METHOD PUBLIC IsFaulted : BOOL
VAR_INPUT
END_VAR
IsFaulted := (State = eGoodULNewStaState.eUnknown OR State = eGoodULNewStaState.eError);
END_METHOD

METHOD PUBLIC IsPalletHoldDownEngaged : BOOL
VAR_INPUT
END_VAR
IsPalletHoldDownEngaged := (GVL_IO.UL_3_XPalletHoldDownRetracted_Engaged AND NOT GVL_IO.UL_3_XPalletHoldDownExtended_Home);
IF (NOT IsPalletHoldDownEngaged) THEN
	Status.GoodUL_3_StatusMsg:= 'Good UL 3: Check Pallet Hold Down Sensors and then hit START';
END_IF
END_METHOD

METHOD PUBLIC IsPalletHoldDownFree : BOOL
VAR_INPUT
END_VAR
IsPalletHoldDownFree := (NOT GVL_IO.UL_3_XPalletHoldDownRetracted_Engaged AND GVL_IO.UL_3_XPalletHoldDownExtended_Home);
IF (NOT IsPalletHoldDownFree) THEN
	Status.GoodUL_3_StatusMsg := 'Good UL 3: Check Pallet Hold Down Sensors and then hit START';
END_IF
END_METHOD

PROPERTY PUBLIC Ready : BOOL
GET
IF (LotsData.Lot.GoodUnloadEnabled) THEN
	Ready := (State = eGoodULNewStaState.eReady);
ELSE
	Ready := (State = eGoodULNewStaState.eDisabledReady); 
END_IF
END_GET
END_PROPERTY

ACTION ResetDwellTimer:
DwellTimer(IN:=FALSE);
END_ACTION

METHOD PUBLIC ResetState : BOOL
VAR_INPUT
END_VAR
State := eGoodULNewStaState.eUnknown;
NextState := eGoodULNewStaState.eUnknown;
END_METHOD

PROPERTY PUBLIC Trigger : BOOL
SET
xTrigger := Trigger;
END_SET
END_PROPERTY

METHOD PUBLIC UpdateLotData : BOOL
VAR_INPUT
END_VAR
IF (PartsData.Status[VUT].Premium) THEN
	LotsData.Lot.CavityCounts[PartsData.Status[VUT].CavityNumber].PremiumCount := LotsData.Lot.CavityCounts[PartsData.Status[VUT].CavityNumber].PremiumCount +1;
ELSIF (PartsData.Status[VUT].Good) THEN
 	LotsData.Lot.CavityCounts[PartsData.Status[VUT].CavityNumber].GoodCount := LotsData.Lot.CavityCounts[PartsData.Status[VUT].CavityNumber].GoodCount + 1;
END_IF
LotsData.Lot.CavityCounts[PartsData.Status[VUT].CavityNumber].TotalCount := LotsData.Lot.CavityCounts[PartsData.Status[VUT].CavityNumber].TotalCount + 1;
 // reject parts shouldn't get here. If this station rejects something (e.g. faults out) then it barrel will go to reject station.
END_METHOD

METHOD PUBLIC UpdatePartData : BOOL
VAR_INPUT
END_VAR
PartsData.Status[VUT].UnloadTime := SYSTEMTIME_TO_STRING(Logging.fbCurrTime.systemTime);
PartsData.Status[VUT].OverallStatus := ePartStatus.eEmpty;
PartsData.Status[VUT].GoodUnload := TRUE;

// we will write data to CSV file over here 
IF (P_TextModeWrite.CurrWriteStep = 0) THEN 
	P_TextModeWrite.VehicleID := VUT;
	P_TextModeWrite.WriteData := TRUE;
END_IF
END_METHOD

PROPERTY PUBLIC VehicleUnderTest : BYTE
GET
VehicleUnderTest := VUT;
END_GET
SET
VUT := VehicleUnderTest;
END_SET
END_PROPERTY

END_FUNCTION_BLOCK

// ---- POUs/GoodULStation_4.TcPOU
FUNCTION_BLOCK PUBLIC GoodULStation_4
VAR_INPUT
END_VAR
VAR_OUTPUT
END_VAR
VAR
	xTrigger :BOOL := FALSE; // triggers processing
	State : eGoodULNewStaState := eGoodULNewStaState.eUnknown;
	NextState : eGoodULNewStaState := eGoodULNewStaState.eUnknown;
	ErrorReturnState : eGoodULNewStaState := eGoodULNewStaState.eUnknown;
	bFirst : BOOL := TRUE;
	VUT : BYTE; //VehicleID Under Station
	DwellTimer : TON;
	StateTimer : TON;
	GoodFullExcess: BYTE := 0;
END_VAR

IF (GVL_IO.MachineEStopped) THEN 
	State := eGoodULNewStaState.eUnknown;
	NextState := eGoodULNewStaState.eUnknown;
	Status.GoodUL_4_StatusMsg:= 'Good UL 4 Sta Unknown, Check AIR, E-STOP and Hit Start';
END_IF

CASE State OF
eGoodULNewStaState.eUnknown:
	Status.GoodUL_4_StatusMsg:= 'Good UL 4 Unknown, Check AIR, E-STOP and Hit Start';
    IF (GVL_IO.MC_XStartPB AND GVL_IO.MC_XAirPressureOK AND GVL_IO.MC_NotEStopped) THEN // wait for start button when powered up or PLC program restarted
		NextState := eGoodULNewStaState.eInit;	   
	END_IF
    

eGoodULNewStaState.eInit:
    Act_KnockPartOFF();
	Act_FreePalletHoldDown();
	ResetDwellTimer();
	NextState := eGoodULNewStaState.eHoming;
	

eGoodULNewStaState.eHoming:
	IF (IsPalletHoldDownFree()) THEN 
         NextState := eGoodULNewStaState.eReady;
	  END_IF
     DwellTimer(IN:=TRUE, PT:= T#10S);
     IF (DwellTimer.Q) THEN
		 ResetDwellTimer();
		 ErrorReturnState:= eGoodULNewStaState.eInit;
		 NextState := eGoodULNewStaState.eError;		 
	 END_IF	

eGoodULNewStaState.eReady:
	IF (xTrigger) THEN
		IF (NOT LotsData.Lot.AutoBaggerEnabled) THEN 
				Stations.fbRoutePlanner.P_GoodUnload_4_NextStaFlag := 5; 
				NextState := eGoodULNewStaState.eSendPalletHoldDownExtend;	
		ELSE
				NextState := eGoodULNewStaState.eCheckChuteCount;	
		END_IF	
		ResetDwellTimer();
	END_IF
	
	IF (NOT LotsData.Lot.GoodUnloadEnabled) THEN
		NextState :=  eGoodULNewStaState.eDisabledReady;	
	END_IF

eGoodULNewStaState.eDisabledReady:

	Act_KnockPartOFF();
	Act_FreePalletHoldDown();
	
    IF (LotsData.Lot.GoodUnloadEnabled) THEN 
		NextState := eGoodULNewStaState.eUnknown; // force the operator to hit the start button if station is enabled.
	END_IF
	
    IF (xTrigger) THEN // vehicles that have been previously commanded to come here before station was disabled 
		Stations.fbRoutePlanner.P_GoodUnload_4_NextStaFlag := 5; // send to reject after this process is complete
		NextState := eGoodULNewStaState.eDepart;
	END_IF
	
	Status.StationStauts[MM_CONST.GOOD_UL_4_STA_HMI_STATE] := OverallStationStatus.eDisabled;
	Status.GoodUL_4_StatusMsg:= 'Good UL1 Disabled and Clear for pallets to move';	

eGoodULNewStaState.eCheckChuteCount:
	IF  (Config.GoodCount2 < LotsData.Lot.QuantityInBag)  THEN
			Stations.fbRoutePlanner.P_GoodUnload_4_NextStaFlag := 5; // send to reject after this process is complete
			NextState := eGoodULNewStaState.eSendPalletHoldDownExtend;	          
 			GoodFullExcess:=0;  			
	ELSE  	
		    GoodFullExcess := GoodFullExcess +1;
			Stations.fbRoutePlanner.P_GoodUnload_4_NextStaFlag := 5; // send to reject after this process is complete
			NextState := eGoodULNewStaState.eDepart;
	END_IF 		
	IF (GoodFullExcess > 5) THEN 
		ErrorReturnState:= eGoodULNewStaState.eCheckChuteCount;		
		Status.GoodUL_4_StatusMsg:= 'No Drop Location for Part!Fix Bagger & Clear Chutes';
		NextState := eGoodULNewStaState.eError;		
    END_IF			


eGoodULNewStaState.eSendPalletHoldDownExtend:
	Act_EngagePalletHoldDown();
	ResetDwellTimer();
	NextState := eGoodULNewStaState.eCheckPalletHoldDownExtended;
	
eGoodULNewStaState.eCheckPalletHoldDownExtended:
   DwellTimer(IN:=TRUE, PT:= T#10S);	
   IF (IsPalletHoldDownEngaged()) THEN
        ResetDwellTimer();	   
		IF(GVL_IO.UL_4_XBarrelPresent (*OR TRUE*)) THEN /// enabled checking Part Present Sensor at Unload stations 051319 NAP
			NextState := eGoodULNewStaState.eKnockOffPart;
        ELSE
			NextState := eGoodULNewStaState.ePalletHoldDownRelease;	
		END_IF        
   END_IF      
   IF (DwellTimer.Q) THEN
		 ResetDwellTimer();
		 ErrorReturnState:= eGoodULNewStaState.eSendPalletHoldDownExtend;
		 NextState := eGoodULNewStaState.eError;		 
	END_IF
  
eGoodULNewStaState.eKnockoffPart:
	Act_KnockPartON();
	UpdateLotData();
	UpdatePartData();
	ResetDwellTimer();
	StateTimer(IN:=FALSE);	
	NextState := eGoodULNewStaState.eCheckPartKnockedOff;

eGoodULNewStaState.eCheckPartKnockedOff:
   StateTimer(IN:=TRUE, PT:= T#200MS);
   	IF (StateTimer.Q) THEN
   //IF (NOT(GVL_IO.UL_4_XBarrelPresent) ) THEN   
	   NextState := eGoodULNewStaState.ePalletHoldDownRelease;
	   Config.GoodCount2 := Config.GoodCount2 + 1;
	   DwellTimer(IN:=FALSE);
	   StateTimer(IN:=FALSE);
   END_IF
   DwellTimer(IN:= TRUE, PT:= T#10S);
   IF (DwellTimer.Q) THEN
	   ResetDwellTimer();
	   ErrorReturnState:= eGoodULNewStaState.eCheckPartKnockedOff;
	   Status.GoodUL_4_StatusMsg:= 'Good UL 4 Remove Part then Hit START';
   	   NextState := eGoodULNewStaState.eError;	
   END_IF   

eGoodULNewStaState.ePalletHoldDownRelease:
    Act_KnockPartOFF();
	Act_FreePalletHoldDown();
    ResetDwellTimer();	
	NextState := eGoodULNewStaState.ePalletHoldDownReleased;

eGoodULNewStaState.ePalletHoldDownReleased:	
	IF (IsPalletHoldDownFree()) THEN         
	    NextState := eGoodULNewStaState.eDepart;
    END_IF
	
   DwellTimer(IN:= TRUE, PT:= T#10S);
   IF (DwellTimer.Q) THEN
	   ResetDwellTimer();
	   ErrorReturnState:= eGoodULNewStaState.ePalletHoldDownRelease;	   
   	   NextState := eGoodULNewStaState.eError;	
   END_IF  
	
	
eGoodULNewStaState.eDepart:
    Stations.fbRoutePlanner.M_NotifyVehStaCmpl(StationIndex:= MM_CONST.GOOD_UL_4_STA, VehicleID := VUT);
	xTrigger := FALSE;
	IF (Stations.fbCycleControl.StopRequested) THEN
		NextState := eGoodULNewStaState.eStopActive;
	ELSE 
		NextState := eGoodULNewStaState.eReady;
    END_IF
	
eGoodULNewStaState.eStopActive:
	IF (NOT Stations.fbCycleControl.StopRequested) THEN
		NextState := eGoodULNewStaState.eInit;
    END_IF
	

eGoodULNewStaState.eError:
	IF (GVL_IO.MC_XStartPB) THEN
		NextState := ErrorReturnState;
		ErrorReturnState := eGoodULNewStaState.eUnknown;
	END_IF

END_CASE

IF (State <> NextState) THEN
	bFirst := TRUE;
	StateTimer(IN:=FALSE);
ELSE
	bFirst := FALSE;
END_IF

State := NextState;
AssignStationStatusForHMI();

ACTION Act_EngagePalletHoldDown:
GVL_IO.UL_4_YPalletHoldDownExtend_Home  := FALSE;
GVL_IO.UL_4_YPalletHoldDownRetract_Engage := TRUE;
END_ACTION

ACTION Act_FreePalletHoldDown:
GVL_IO.UL_4_YPalletHoldDownExtend_Home := TRUE;
GVL_IO.UL_4_YPalletHoldDownRetract_Engage := FALSE;
END_ACTION

ACTION Act_KnockPartOFF:
GVL_IO.UL_4_YRejectPushExtend := FALSE;
GVL_IO.UL_4_YRejectPushRetract := TRUE;
END_ACTION

ACTION Act_KnockPartON:
GVL_IO.UL_4_YRejectPushExtend := TRUE;
GVL_IO.UL_4_YRejectPushRetract := FALSE;
END_ACTION

METHOD PUBLIC AssignStationStatusForHMI : BOOL
VAR_INPUT
END_VAR
Status.StationsState[MM_CONST.GOOD_UL_4_STA_HMI_STATE] := State;
IF (NOT LotsData.Lot.GoodUnloadEnabled) THEN
	Status.StationStauts[MM_CONST.GOOD_UL_4_STA_HMI_STATE] := OverallStationStatus.eDisabled;
ELSE 
	CASE State OF 
	
	eGoodULNewStaState.eUnknown,eGoodULNewStaState.eError:
		Status.StationStauts[MM_CONST.GOOD_UL_4_STA_HMI_STATE] := OverallStationStatus.eError;
		
    eGoodULNewStaState.eInit,
	eGoodULNewStaState.eHoming:
	    Status.StationStauts[MM_CONST.GOOD_UL_4_STA_HMI_STATE] := OverallStationStatus.eHoming;
	
	eGoodULNewStaState.eReady,eGoodULNewStaState.eWaitForVehicleTrigger:
	     Status.StationStauts[MM_CONST.GOOD_UL_4_STA_HMI_STATE] := OverallStationStatus.eWaitingForParts;
		 
	eGoodULNewStaState.eDwell,
	eGoodULNewStaState.eSendPalletHoldDownExtend,
	eGoodULNewStaState.eCheckPalletHoldDownExtended,
	eGoodULNewStaState.ePalletReleaseExtend,
	eGoodULNewStaState.ePalletReleaseExtended,
	eGoodULNewStaState.eKnockoffPart,
	eGoodULNewStaState.eKnockoffExtended,
	eGoodULNewStaState.eCheckPartKnockedOff,
	eGoodULNewStaState.ePalletHoldDownRelease,
	eGoodULNewStaState.ePalletHoldDownReleased:
	    Status.StationStauts[MM_CONST.GOOD_UL_4_STA_HMI_STATE] := OverallStationStatus.eRunning;
	
	eGoodULNewStaState.eStopActive:
	    Status.StationStauts[MM_CONST.GOOD_UL_4_STA_HMI_STATE] := OverallStationStatus.eCycleStop;
    	
	
    ELSE;	
	END_CASE
END_IF
END_METHOD

METHOD PUBLIC ClearVehicleTrigger : BOOL
VAR_INPUT
END_VAR
xTrigger := FALSE;
END_METHOD

METHOD PUBLIC IsFaulted : BOOL
VAR_INPUT
END_VAR
IsFaulted := (State = eGoodULNewStaState.eUnknown OR State = eGoodULNewStaState.eError);
END_METHOD

METHOD PUBLIC IsPalletHoldDownEngaged : BOOL
VAR_INPUT
END_VAR
IsPalletHoldDownEngaged := (GVL_IO.UL_4_XPalletHoldDownRetracted_Engaged AND NOT GVL_IO.UL_4_XPalletHoldDownExtended_Home);
IF (NOT IsPalletHoldDownEngaged) THEN
	Status.GoodUL_4_StatusMsg:= 'Good UL 4: Check Pallet Hold Down Sensors and then hit START';
END_IF
END_METHOD

METHOD PUBLIC IsPalletHoldDownFree : BOOL
VAR_INPUT
END_VAR
IsPalletHoldDownFree := (NOT GVL_IO.UL_4_XPalletHoldDownRetracted_Engaged AND GVL_IO.UL_4_XPalletHoldDownExtended_Home);
IF (NOT IsPalletHoldDownFree) THEN
	Status.GoodUL_4_StatusMsg := 'Good UL 4: Check Pallet Hold Down Sensors and then hit START';
END_IF
END_METHOD

PROPERTY PUBLIC Ready : BOOL
GET
IF (LotsData.Lot.GoodUnloadEnabled) THEN
	Ready := (State = eGoodULNewStaState.eReady);
ELSE
	Ready := (State = eGoodULNewStaState.eDisabledReady); 
END_IF
END_GET
END_PROPERTY

ACTION ResetDwellTimer:
DwellTimer(IN:=FALSE);
END_ACTION

METHOD PUBLIC ResetState : BOOL
VAR_INPUT
END_VAR
State := eGoodULNewStaState.eUnknown;
NextState := eGoodULNewStaState.eUnknown;
END_METHOD

PROPERTY PUBLIC Trigger : BOOL
SET
xTrigger := Trigger;
END_SET
END_PROPERTY

METHOD PUBLIC UpdateLotData : BOOL
VAR_INPUT
END_VAR
IF (PartsData.Status[VUT].Premium) THEN
	LotsData.Lot.CavityCounts[PartsData.Status[VUT].CavityNumber].PremiumCount := LotsData.Lot.CavityCounts[PartsData.Status[VUT].CavityNumber].PremiumCount +1;
ELSIF (PartsData.Status[VUT].Good) THEN
 	LotsData.Lot.CavityCounts[PartsData.Status[VUT].CavityNumber].GoodCount := LotsData.Lot.CavityCounts[PartsData.Status[VUT].CavityNumber].GoodCount + 1;
END_IF
LotsData.Lot.CavityCounts[PartsData.Status[VUT].CavityNumber].TotalCount := LotsData.Lot.CavityCounts[PartsData.Status[VUT].CavityNumber].TotalCount + 1;
 // reject parts shouldn't get here. If this station rejects something (e.g. faults out) then it barrel will go to reject station.
END_METHOD

METHOD PUBLIC UpdatePartData : BOOL
VAR_INPUT
END_VAR
PartsData.Status[VUT].UnloadTime := SYSTEMTIME_TO_STRING(Logging.fbCurrTime.systemTime);
PartsData.Status[VUT].OverallStatus := ePartStatus.eEmpty;
PartsData.Status[VUT].GoodUnload := TRUE;

// we will write data to CSV file over here 
IF (P_TextModeWrite.CurrWriteStep = 0) THEN 
	P_TextModeWrite.VehicleID := VUT;
	P_TextModeWrite.WriteData := TRUE;
END_IF
END_METHOD

PROPERTY PUBLIC VehicleUnderTest : BYTE
GET
VehicleUnderTest := VUT;
END_GET
SET
VUT := VehicleUnderTest;
END_SET
END_PROPERTY

END_FUNCTION_BLOCK

// ---- POUs/RejectStation.TcPOU
FUNCTION_BLOCK PUBLIC RejectStation
VAR_INPUT
END_VAR
VAR_OUTPUT
END_VAR
VAR
	xTrigger :BOOL := FALSE; // triggers processing
	State : eRejectStaState := eRejectStaState.eUnknown;
	NextState : eRejectStaState := eRejectStaState.eUnknown;
	ErrorReturnState : eRejectStaState := eRejectStaState.eUnknown;
	bFirst : BOOL := TRUE;
	VUT : BYTE; //VehicleID Under Station
	DwellTimer : TON;
	StateTimer : TON;
END_VAR

IF (GVL_IO.MachineEStopped) THEN 
	State := eRejectStaState.eUnknown;
	NextState := eRejectStaState.eUnknown;
	Status.RejectStatusMsg:= 'RejectSta Unknown, Check AIR, E-STOP and Hit Start';
END_IF

CASE State OF
eRejectStaState.eUnknown:
	Status.RejectStatusMsg:= 'RejectSta Unknown, Check AIR, E-STOP and Hit Start';
    IF (GVL_IO.MC_XStartPB AND GVL_IO.MC_XAirPressureOK AND GVL_IO.MC_NotEStopped) THEN // wait for start button when powered up or PLC program restarted
		NextState := eRejectStaState.eInit;	   
	END_IF
    

eRejectStaState.eInit:
    Act_KnockPartOFF();
	Act_FreePalletHoldDown();
	ResetDwellTimer();
	NextState := eRejectStaState.eHoming;
	

eRejectStaState.eHoming:
	IF (IsPalletHoldDownFree()) THEN 
         NextState := eRejectStaState.eReady;
	  END_IF
     DwellTimer(IN:=TRUE, PT:= T#10S);
     IF (DwellTimer.Q) THEN
		 ResetDwellTimer();
		 ErrorReturnState:= eRejectStaState.eInit;
		 NextState := eRejectStaState.eError;		 
	 END_IF	

eRejectStaState.eReady:
	IF (xTrigger) THEN
		NextState := eRejectStaState.eSendPalletHoldDownExtend;		
		ResetDwellTimer();
	END_IF

eRejectStaState.eSendPalletHoldDownExtend:
	Act_EngagePalletHoldDown();
	ResetDwellTimer();
	NextState := eRejectStaState.eCheckPalletHoldDownExtended;
	
eRejectStaState.eCheckPalletHoldDownExtended:
   DwellTimer(IN:=TRUE, PT:= T#10S);	
   IF (IsPalletHoldDownEngaged()) THEN
        ResetDwellTimer();	   
		IF(GVL_IO.RJ_XPartPresent OR TRUE) THEN         //added Turnkey shop sensor not adjusted
			NextState := eRejectStaState.eKnockOffPart;
			ResetDwellTimer();
        ELSE
			NextState := eRejectStaState.ePalletHoldDownRelease;	
		END_IF        
   END_IF      
   IF (DwellTimer.Q) THEN
		 ResetDwellTimer();
		 ErrorReturnState:= eRejectStaState.eSendPalletHoldDownExtend;
		 NextState := eRejectStaState.eError;		 
	END_IF
  
eRejectStaState.eKnockoffPart:
	Act_KnockPartON();
	UpdateLotData();
	UpdatePartData();
    DwellTimer(IN:=TRUE, PT:= T#250MS);
    IF (DwellTimer.Q) THEN 
		NextState := eRejectStaState.eCheckPartKnockedOff;
		ResetDwellTimer();
	END_IF;

eRejectStaState.eCheckPartKnockedOff:
   IF (NOT(GVL_IO.RJ_XPartPresent) ) THEN   /// until Bonnie can ajust sensor
	   NextState := eRejectStaState.ePalletHoldDownRelease;
	   DwellTimer(IN:=FALSE);
	   StateTimer(IN:=FALSE);
   END_IF
   DwellTimer(IN:= TRUE, PT:= T#10S);
   IF (DwellTimer.Q) THEN
	   ResetDwellTimer();
	   ErrorReturnState:= eRejectStaState.eCheckPartKnockedOff;
	   Status.RejectStatusMsg:= 'Reject Remove Part then Hit START';
   	   NextState := eRejectStaState.eError;	
   END_IF   

eRejectStaState.ePalletHoldDownRelease:
    Act_KnockPartOFF();
	Act_FreePalletHoldDown();
    ResetDwellTimer();	
	NextState := eRejectStaState.ePalletHoldDownReleased;

eRejectStaState.ePalletHoldDownReleased:	
	IF (IsPalletHoldDownFree()) THEN         
	    NextState := eRejectStaState.eDepart;
    END_IF
	
   DwellTimer(IN:= TRUE, PT:= T#10S);
   IF (DwellTimer.Q) THEN
	   ResetDwellTimer();
	   ErrorReturnState:= eRejectStaState.ePalletHoldDownRelease;	   
   	   NextState := eRejectStaState.eError;	
   END_IF  
	
	
eRejectStaState.eDepart:
    Stations.fbRoutePlanner.M_NotifyVehStaCmpl(StationIndex:= MM_CONST.REJECT_ULOAD_STA, VehicleID := VUT);
	xTrigger := FALSE;
	IF (Stations.fbCycleControl.StopRequested) THEN
		NextState := eRejectStaState.eStopActive;
	ELSE 
		NextState := eRejectStaState.eReady;
    END_IF
	
eRejectStaState.eStopActive:
	IF (NOT Stations.fbCycleControl.StopRequested) THEN
		NextState := eRejectStaState.eReady;
    END_IF
	

eRejectStaState.eError:
	IF (GVL_IO.MC_XStartPB) THEN
		NextState := ErrorReturnState;
		ErrorReturnState := eRejectStaState.eUnknown;
	END_IF

END_CASE

IF (State <> NextState) THEN
	bFirst := TRUE;
	StateTimer(IN:=FALSE);
ELSE
	bFirst := FALSE;
END_IF

State := NextState;
AssignStationStatusForHMI();

ACTION Act_EngagePalletHoldDown:
GVL_IO.RJ_YPalletHoldDownExtend_Home  := FALSE;
GVL_IO.RJ_YPalletHoldDownRetract_Engage := TRUE;
END_ACTION

ACTION Act_FreePalletHoldDown:
GVL_IO.RJ_YPalletHoldDownExtend_Home := TRUE;
GVL_IO.RJ_YPalletHoldDownRetract_Engage := FALSE;
END_ACTION

ACTION Act_KnockPartOFF:
	GVL_IO.RJ_YRejectPushExtend := FALSE;
	GVL_IO.RJ_YRejectPushRetract := TRUE;
END_ACTION

ACTION Act_KnockPartON:
	GVL_IO.RJ_YRejectPushExtend := TRUE;
	GVL_IO.RJ_YRejectPushRetract := FALSE;
END_ACTION

METHOD PUBLIC AssignStationStatusForHMI : BOOL
VAR_INPUT
END_VAR
Status.StationsState[MM_CONST.REJECT_ULOAD_STA_HMI_STATE] := State;
IF (NOT LotsData.Lot.RejectUnloadEnabled) THEN
	Status.StationStauts[MM_CONST.REJECT_ULOAD_STA_HMI_STATE] := OverallStationStatus.eDisabled;
ELSE 
	CASE State OF 
	
	eRejectStaState.eUnknown,eRejectStaState.eError:
		Status.StationStauts[MM_CONST.REJECT_ULOAD_STA_HMI_STATE] := OverallStationStatus.eError;
		
    eRejectStaState.eInit,
	eRejectStaState.eHoming:
	    Status.StationStauts[MM_CONST.REJECT_ULOAD_STA_HMI_STATE] := OverallStationStatus.eHoming;
	
	eRejectStaState.eReady,eRejectStaState.eWaitForVehicleTrigger:
	     Status.StationStauts[MM_CONST.REJECT_ULOAD_STA_HMI_STATE] := OverallStationStatus.eWaitingForParts;
		 
	eRejectStaState.eDwell,
	eRejectStaState.eSendPalletHoldDownExtend,
	eRejectStaState.eCheckPalletHoldDownExtended,
	eRejectStaState.ePalletReleaseExtend,
	eRejectStaState.ePalletReleaseExtended,
	eRejectStaState.eKnockoffPart,
	eRejectStaState.eKnockoffExtended,
	eRejectStaState.eCheckPartKnockedOff,
	eRejectStaState.ePalletHoldDownRelease,
	eRejectStaState.ePalletHoldDownReleased:
	    Status.StationStauts[MM_CONST.REJECT_ULOAD_STA_HMI_STATE] := OverallStationStatus.eRunning;
	
	eRejectStaState.eStopActive:
	    Status.StationStauts[MM_CONST.REJECT_ULOAD_STA_HMI_STATE] := OverallStationStatus.eCycleStop;
    	
	
    ELSE;	
	END_CASE
END_IF
END_METHOD

METHOD PUBLIC ClearVehicleTrigger : BOOL
VAR_INPUT
END_VAR
xTrigger := FALSE;
END_METHOD

METHOD PUBLIC IsFaulted : BOOL
VAR_INPUT
END_VAR
IsFaulted := (State = eRejectStaState.eUnknown OR State = eRejectStaState.eError);
END_METHOD

METHOD PUBLIC IsPalletHoldDownEngaged : BOOL
VAR_INPUT
END_VAR
IsPalletHoldDownEngaged := (GVL_IO.RJ_XPalletHoldDownRetracted_Engaged AND NOT GVL_IO.RJ_XPalletHoldDownExtended_Home);
IF (NOT IsPalletHoldDownEngaged) THEN
	Status.RejectStatusMsg:= 'Reject: Check Pallet Hold Down Sensors and then hit START';
END_IF
END_METHOD

METHOD PUBLIC IsPalletHoldDownFree : BOOL
VAR_INPUT
END_VAR
IsPalletHoldDownFree := (NOT GVL_IO.RJ_XPalletHoldDownRetracted_Engaged AND GVL_IO.RJ_XPalletHoldDownExtended_Home);
IF (NOT IsPalletHoldDownFree) THEN
	Status.RejectStatusMsg:= 'Reject: Check Pallet Hold Down Sensors and then hit START';
END_IF
END_METHOD

PROPERTY PUBLIC Ready : BOOL
GET
Ready := (State = eRejectStaState.eReady);
END_GET
END_PROPERTY

ACTION ResetDwellTimer:
DwellTimer(IN:=FALSE);
END_ACTION

METHOD PUBLIC ResetState : BOOL
VAR_INPUT
END_VAR
State := eRejectStaState.eUnknown;
NextState := eRejectStaState.eUnknown;
END_METHOD

PROPERTY PUBLIC Trigger : BOOL
SET
xTrigger := Trigger;
END_SET
END_PROPERTY

METHOD PUBLIC UpdateLotData : BOOL
VAR_INPUT
END_VAR
IF (PartsData.Status[VUT].OverallStatus <> ePartStatus.eEmpty) THEN
	LotsData.Lot.CavityCounts[PartsData.Status[VUT].CavityNumber].BadCount := LotsData.Lot.CavityCounts[PartsData.Status[VUT].CavityNumber].BadCount +1;
	LotsData.Lot.CavityCounts[PartsData.Status[VUT].CavityNumber].TotalCount := LotsData.Lot.CavityCounts[PartsData.Status[VUT].CavityNumber].TotalCount + 1;
END_IF
END_METHOD

METHOD PUBLIC UpdatePartData : BOOL
VAR_INPUT
END_VAR
PartsData.Status[VUT].RejectUnloadTime := SYSTEMTIME_TO_STRING(Logging.fbCurrTime.systemTime);
IF (PartsData.Status[VUT].OverallStatus <> ePartStatus.eEmpty) THEN
	IF (P_TextModeWrite.CurrWriteStep = 0) THEN (* if resource not ready, we will skip this part*)
    P_TextModeWrite.VehicleID := VUT;
	P_TextModeWrite.WriteData := TRUE;
	END_IF 
END_IF
PartsData.Status[VUT].OverallStatus := ePartStatus.eEmpty;

// we will write data to CSV file over here
END_METHOD

PROPERTY PUBLIC VehicleUnderTest : BYTE
GET
VehicleUnderTest := VUT;
END_GET
SET
VUT := VehicleUnderTest;
END_SET
END_PROPERTY

END_FUNCTION_BLOCK

// ---- POUs/BurnOffStation.TcPOU
FUNCTION_BLOCK BurnOffStation
VAR_INPUT
END_VAR
VAR_OUTPUT
END_VAR
VAR
	HeaterONTimer : TON;
	BlowerOFFTimer : TON;
	PrevRunning, CurrRunning : BOOL := FALSE;
	StartFromReset, StopAfterEStop : BOOL:=FALSE;	
	BlowerEnable: BOOL := FALSE;
	HeatEnable: BOOL := FALSE;
	PIDEnable: BOOL := FALSE;
	nErrorPIDStatus : UINT;
	PIDOutput : LREAL;
	VoltOutReal : LREAL;
	fbBurnoffPID :FB_BasicPID;
	// Temperature needs to be divided by 10 after reading from the TC card
	fProcessValue: LREAL := 0;
END_VAR

fProcessValue := GVL_IO.BU_Temperature/10;	
STATUS.BurnOffTemperature := LREAL_TO_DINT(fProcessValue);

IF (NOT LotsData.Lot.BurnOffEnabled OR STATIONS.fbMMMonitor.IsMMJammed OR Stations.fbCycleControl.StopRequested OR GVL_IO.MachineEStopped OR Status.BurnOffIdle) THEN
	GVL_IO.BU_HeatCntl := 0;
	GVL_IO.BU_BlowCntl := 0;
ELSE 
	// set the blower setpoint from the User configuration in HMI
	GVL_IO.BU_BlowCntl := REAL_TO_INT(CONFIG.BU_BLOWER_SETPOINT/100*32000); 
	IF ( GVL_IO.BU_BlowCntl > 32000) THEN
		GVL_IO.BU_BlowCntl := 32000;
	END_IF
	// set the heater output based on proporational control with limits 
	fbBurnoffPID (fSetpointValue:= LotsData.Lot.BurnOffTemp +25,
					fActualValue := fProcessValue,
					bReset := FALSE,
					fCtrlCycleTime:=TIME_TO_LREAL(T#500MS),
					fKp:=1000,
					fTn:=0,//TIME_TO_LREAL(T#20MS),
					fTv:=0,//TIME_TO_LREAL(T#200MS),
					fTd:=0,//TIME_TO_LREAL(T#100MS),
					fCtrlOutput =>PIDOutput,
					nErrorStatus => nErrorPIDStatus);			
	        
	IF (PIDOutput>32767) THEN
		PIDOutput := 32767; // full heat, a value of  0.5V will be sent to heater control element. We don't want to heater element too hot
	END_IF
	IF (PIDOutput<0) THEN
		PIDOutput := 0; // No heat, a value of 0 V will be sent to heater control element
	END_IF       
		GVL_IO.BU_HeatCntl := LREAL_TO_INT(PIDOutput); // Write this data out to the Analog Output Card
END_IF

AssignStationStatusForHMI();

METHOD PUBLIC AssignStationStatusForHMI : BOOL
VAR_INPUT
END_VAR
Status.StationsState[MM_CONST.BURNOFF_STA_HMI_STATE] := BOOL_TO_INT(HeatEnable);
IF (LotsData.Lot.BurnOffEnabled) THEN
	IF ((ABS(fProcessValue - LotsData.Lot.BurnOffTemp)) > 25) THEN  // to replace with actual setpoint from user screen
    	Status.StationStauts[MM_CONST.BURNOFF_STA_HMI_STATE] := OverallStationStatus.eHoming;
		Status.BurnOffStatusMsg:= 'Not At Temperature!';
		Status.StationInfoString[MM_CONST.BURNOFF_STA_HMI_STATE] := 'Check BurnOff Leister Powered ON';
	ELSE	
		Status.StationStauts[MM_CONST.BURNOFF_STA_HMI_STATE] := OverallStationStatus.eRunning;
		Status.BurnOffStatusMsg := 'At Temperature';
		Status.StationInfoString[MM_CONST.BURNOFF_STA_HMI_STATE] := '';
	END_IF
END_IF
END_METHOD

PROPERTY PUBLIC IsAtTemperature : BOOL
GET
IsAtTemperature := TRUE;//(Status.StationStauts[MM_CONST.BURNOFF_STA_HMI_STATE] = OverallStationStatus.eRunning);
END_GET
SET
END_SET
END_PROPERTY

END_FUNCTION_BLOCK

// ---- POUs/CapInsertStation_Old.TcPOU
FUNCTION_BLOCK PUBLIC CapInsertStation_Old
VAR_INPUT
END_VAR
VAR_OUTPUT
END_VAR
VAR
	xTrigger :BOOL := FALSE; // triggers processing
	State : eCapInsertStaState := eCapInsertStaState.eUnknown;
	NextState : eCapInsertStaState := eCapInsertStaState.eUnknown;
	bFirst : BOOL := TRUE;
	VUT : BYTE; //VehicleID Under Station
	DwellTimer : TON;		
	StateTimer : TON;
	PartPresentTimer : TON;
	CapInstallRetries : BYTE :=0;
	CapPickUpRetries : BYTE := 0;
END_VAR

//////////////////// ESTOP TO STATION DISABLED
// If Cap Station is disabled, then we want to make sure that we have the SMAC homed and not in the way of barrels
// we also want to check if the pallet hold downs and center pins are in the correct position
// if all above conditions are true, then we want to wait in a station disabled ready state
////////////////// STATION DISABLED - STATION ENABLED
// We have to go pick up a cap and not bring the station in ready condition until cap
// is picked up
/////////////////////// STATION ENABLED - STATION DISABLED
// We have to let go of the vacuum in the tool, and set Next State to Station Disabled Ready
//////////////////////// ESTOP- STATION ENABLED
//// Follow all the logic to get the station ready

IF (GVL_IO.MachineEStopped) THEN 
	State := eCapInsertStaState.eUnknown;
	NextState := eCapInsertStaState.eUnknown;
	Status.CapStatusMsg:= 'CapSta Unknown State, Check AIR, E-STOP and Hit Start';
END_IF

CASE State OF

eCapInsertStaState.eUnknown:
	   IF (GVL_IO.MC_XStartPB AND GVL_IO.MC_XAirPressureOK AND GVL_IO.MC_NotEStopped) THEN // wait for start button when powered up or PLC program restarted
			NextState := eCapInsertStaState.eSMACMtrSendHome;	   
	   END_IF
	GVL_IO.CP_YEscapeWallCylinderExtend:= FALSE;
	GVL_IO.CP_YEscapeWallCylinderRetract := TRUE;
	GVL_IO.CP_YToolVacuumON := FALSE;
	GVL_IO.CP_YToolVacuumOFF := FALSE;	
	GVL_IO.CP_YEscapementToBowl:= FALSE; /// now we have a center OFF valve, turning both valves off will result in air getting dumped	
	GVL_IO.CP_YEscapementToPick:= FALSE;
	StateTimer(IN:=TRUE, PT:= T#9.5S); // give a message out every 10 seconds
	IF (StateTimer.Q) THEN
		Logging.fbEventMsg.SendEventMsg(MsgClass := TCEVENTCLASS_STATEINFO, EventID:= Logging.ID_CP_Unknown, SourceID:= Logging.SrcCapPOU);
		StateTimer(IN:=FALSE);
	END_IF
	
	//Status.StationInfoString[MM_CONST.CAP_STA_HMI_STATE] := '';
	//Status.StationStatusString[MM_CONST.CAP_STA_HMI_STATE] := '';

eCapInsertStaState.eSMACMtrSendHome:
	GVL_IO.CP_YSMAC0 := FALSE;
	GVL_IO.CP_YSMAC1 := TRUE;
	GVL_IO.CP_YSMAC2 := TRUE;
	GVL_IO.CP_YSMAC3 := FALSE;
	DwellTimer(IN:=TRUE, PT:= T#100MS);	
	IF (DwellTimer.Q) THEN
		GVL_IO.CP_YSMAC3 := TRUE; // rising edge to trigger the selected SMAC routine every 5 seconds
		DwellTimer(IN:=FALSE);
		NextState := eCapInsertStaState.eSMACMtrCheckHomed;
	END_IF

eCapInsertStaState.eSMACMtrCheckHomed:
	DwellTimer (IN:= TRUE, PT:= T#250MS);
	IF (DwellTimer.Q) THEN
		 IF (GVL_IO.CP_XSmac2) THEN
		NextState := eCapInsertStaState.eInit;
		GVL_IO.CP_YSMAC3 := FALSE;
		DwellTimer(IN:=FALSE);
		END_IF		
	END_IF
    
	StateTimer(IN:=TRUE, PT:= T#10S); // give a message out every 10 seconds
	IF (StateTimer.Q) THEN
		Logging.fbEventMsg.SendEventMsg(MsgClass := TCEVENTCLASS_STATEINFO, EventID:= Logging.ID_CP_MtrCheckHome, SourceID:= Logging.SrcCapPOU);
		StateTimer(IN:=FALSE);		
		NextState:= eCapInsertStaState.eUnknown; // Operator check what the problem is and then hit the start button again
		GVL_IO.CP_YSMAC3 := FALSE;
		Status.CapStatusMsg:= 'Could not home SMAC, check if SMAC is ON !!';
	END_IF

eCapInsertStaState.eInit:
         GVL_IO.CP_YEscapeWallCylinderExtend:= FALSE;
		 GVL_IO.CP_YEscapeWallCylinderRetract := TRUE; /// we want to check if there is a cap present in the escapement, so need to extend the wall.
		 GVL_IO.CP_YPalletHoldDownExtend := FALSE;
		 GVL_IO.CP_YPalletHoldDownRetract := TRUE;
		 GVL_IO.CP_YBarellCenterPinExtend := FALSE;
		 GVL_IO.CP_YBarellCenterPinRetract := TRUE;
		 GVL_IO.CP_YToolVacuumOFF:= FALSE;
		 GVL_IO.CP_YToolVacuumON:= TRUE; // don't know if vacuum needs to be on, but doesn't hurt to keep it on for 1.5 seconds
		 GVL_IO.CP_YEscapementToBowl := FALSE; // do not move the escapement cyclinder anywhere 
		 GVL_IO.CP_YEscapementToPick := FALSE; // do not move escapement until we read the state of the part presence sensors in tool and escapement
         DwellTimer(IN:= TRUE, PT:= T#1.5S);
		 IF (DwellTimer.Q) THEN
			 DwellTimer(IN:=FALSE);
			 NextState:= eCapInsertStaState.eHoming; 
		 END_IF
			
eCapInsertStaState.eHoming:	
	IF (GVL_IO.CP_XPalletHoldDownHome AND NOT GVL_IO.CP_XPalletHoldDownExtended 
           AND GVL_IO.CP_XSmac2 (*AND GVL_IO.CP_XBarellCenterPinRetracted AND NOT GVL_IO.CP_XBarellCenterPinExtended*) ) THEN  
		   NextState := eCapInsertStaState.eDetermineEscapementPos;	
           IF (NOT LotsData.Lot.CapInsertEnabled) THEN
				NextState :=  eCapInsertStaState.eDisabledReady;
           END_IF 	   
		   DwellTimer(IN:=FALSE);
	END_IF
	StateTimer(IN:=TRUE, PT:= T#10S); // give a message out every 10 seconds
	IF (StateTimer.Q) THEN
		Logging.fbEventMsg.SendEventMsg(MsgClass := TCEVENTCLASS_STATEINFO, EventID:= Logging.ID_CP_AllCheckHome, SourceID:= Logging.SrcCapPOU);
		StateTimer(IN:=FALSE);		
		NextState:= eCapInsertStaState.eUnknown; // Operator check what the problem is and then hit the start button again
		Status.CapStatusMsg:= 'Pallet Hold Down NOT HOME check Cylinders!!';
	END_IF

eCapInsertStaState.eDisabledReady:
	GVL_IO.CP_YToolVacuumOFF:= TRUE;
	GVL_IO.CP_YToolVacuumON:= FALSE;
	IF (LotsData.Lot.CapInsertEnabled) THEN 
		NextState := eCapInsertStaState.eUnknown; // force the operator to hit the start button if station is enabled.
	END_IF
	IF (xTrigger) THEN // vehicles that have been previously commanded to come here before station was disabled 
		NextState := eCapInsertStaState.eDepart;
	END_IF
	Status.CapStatusMsg:= 'Cap Station Disabled, but clear for pallets to move!!';

eCapInsertStaState.eDetermineEscapementPos:

	// First check where the escapement cylinder is located. 
            // If escapement cylinder is at bowl, and if the part present in tool sensor is ON, then we have a part in the tool. We can declare that cap is picked up. 
            // If escapement cyclinder is at bowl, and if the part present in tool sensor is OFF, then we have to wait for a part to be present in the escapement from the bowl feeder
            // If escapment cylinder is at pick location, and there is a part in the tool sensor as well as the part in the escapement, then we part underneath that needs to be picked up by SMAC
			// If escapment cyclinder is at pick location, and there is a part in the tool sensor and no part in the escapement, then we can declare that the cap is picked up.
            // If the escapement is at the pick location, and there is a no part in the tool sensor and no part in the escapement, send the escapement cylinder to the bowl 
            // If the escapement position is undetermined, then if there is no part in the tool and no part in the escapement, send escapement back to bowl
            // If the escapement position is undetermined and if there is a part in the tool and not one in the escapement, then declare that cap is picked up
            // If the escapement position is undetermined and if there is no part in the tool and part is present in escapement, move the part to be picked up
            // If the escapement position is undetermined and if there is a part in the tool and a part in the escapement, then call the operator !!!  
            
			IF (GVL_IO.CP_XEscapementAtBowl AND NOT GVL_IO.CP_XEscapementAtPickUp) THEN // escapement at the bowl
				IF (GVL_IO.CP_XVacuumCapPicked) THEN // we have a part in the tool..
					NextState := eCapInsertStaState.eSendEscapementToBowlNext; // this will pressurize the valves and then wait for vehicle trigger
				ELSE // we have to fetch a part from the bowl location
					NextState:= eCapInsertStaState.eSendEscapementToBowl;
                END_IF
			ELSIF (NOT GVL_IO.CP_XEscapementAtBowl AND GVL_IO.CP_XEscapementAtPickUp) THEN // at the pick location 
				IF (GVL_IO.CP_XVacuumCapPicked AND GVL_IO.CP_XCapPresentEscapment) THEN //we have to pick up this part with the SMAC
					NextState := eCapInsertStaState.eSendEscapementToPick;
				ELSIF(GVL_IO.CP_XVacuumCapPicked AND NOT GVL_IO.CP_XCapPresentEscapment) THEN
				     NextState := eCapInsertStaState.eSendEscapementToBowlNext; // this will pressurize the valves and then wait for vehicle trigger
				ELSIF (NOT GVL_IO.CP_XVacuumCapPicked AND NOT GVL_IO.CP_XCapPresentEscapment) THEN
					NextState:= eCapInsertStaState.eSendEscapementToBowl;
				ELSE
                    NextState := eCapInsertStaState.eUnknown; //send message to HMI over here .. something is wrong with the sensor 
					Status.CapStatusMsg:= 'Check sensor for Cap detection!!';
				END_IF
            ELSE // undetermined location  
				IF (NOT GVL_IO.CP_XVacuumCapPicked AND NOT 	GVL_IO.CP_XCapPresentEscapment) THEN
					NextState:= eCapInsertStaState.eSendEscapementToBowl;
				ELSIF(GVL_IO.CP_XVacuumCapPicked AND NOT GVL_IO.CP_XCapPresentEscapment) THEN
                    NextState := eCapInsertStaState.eSendEscapementToBowlNext; // this will pressurize the valves and then wait for vehicle trigger
				ELSIF(NOT GVL_IO.CP_XVacuumCapPicked AND GVL_IO.CP_XCapPresentEscapment) THEN
 	                NextState := eCapInsertStaState.eSendEscapementToPick;
                ELSIF ( GVL_IO.CP_XVacuumCapPicked AND GVL_IO.CP_XCapPresentEscapment) THEN
                    NextState := eCapInsertStaState.eUnknown; //send message to HMI over here 	
                    Status.CapStatusMsg:= 'Clear CAPS from the Escapement!!';			
                END_IF
			END_IF
	
eCapInsertStaState.eReady: // we need to bypass this state because we added the complex determination of next state from above
	IF (NOT GVL_IO.CP_XPalletHoldDownHome OR GVL_IO.CP_XPalletHoldDownExtended) THEN
		   NextState := eCapInsertStaState.eInit;		   
	  END_IF
	  GVL_IO.CP_YToolVacuumOFF:= FALSE;
	  GVL_IO.CP_YToolVacuumON:= TRUE;
	  DwellTimer(IN:= TRUE, PT:= T#250MS);
	  IF (DwellTimer.Q) THEN
		  DwellTimer(IN:=FALSE);
		  IF (GVL_IO.CP_XVacuumCapPicked) THEN //Cap Already Present 
		  	 NextState := eCapInsertStaState.eWaitForVehicleTrigger;
	      ELSE
			  NextState := eCapInsertStaState.eSendEscapementToBowl;               
			 GVL_IO.CP_YToolVacuumOFF:= TRUE;
		     GVL_IO.CP_YToolVacuumON:= FALSE;
	  	  END_IF	  
	  END_IF
	  

eCapInsertStaState.eSendEscapementToBowl:
	GVL_IO.CP_YToolVacuumOFF:= TRUE;
	  GVL_IO.CP_YToolVacuumON:= FALSE;
    GVL_IO.CP_YEscapementToBowl := TRUE;
	GVL_IO.CP_YEscapementToPick := FALSE;
	IF (GVL_IO.CP_XEscapementAtBowl AND NOT GVL_IO.CP_XEscapementAtPickUp) THEN
    	NextState:= eCapInsertStaState.eEscapementAtBowl; 	
	END_IF	
	StateTimer(IN:=TRUE, PT:= T#5S);
	IF (StateTimer.Q) THEN
		NextState:= eCapInsertStaState.eUnknown;
		Logging.fbEventMsg.SendEventMsg(MsgClass := TCEVENTCLASS_STATEINFO, EventID:= Logging.ID_CP_CheckEscapeCylinders, SourceID:= Logging.SrcCapPOU);
		StateTimer(IN:=FALSE);
		Status.CapStatusMsg:= 'Escapement Did Not reach Bowl, Clear Caps!!';
	END_IF

eCapInsertStaState.eEscapementAtBowl:
  IF (GVL_IO.CP_XCapPresentEscapment) THEN
		PartPresentTimer(IN:= TRUE, PT:= T#100MS); // wait for part to be fully pushed against the back wall
		IF (PartPresentTimer.Q) THEN
			PartPresentTimer(IN:=FALSE);
			NextState := eCapInsertStaState.eSendEscapementToPick;
		END_IF
	ELSE
		PartPresentTimer(IN:=FALSE); //Reset the part present timer here
	END_IF 	

	StateTimer(IN:=TRUE, PT:= T#10S); // give a message out every 10 seconds, hang out here indefinitely to wait for Parts to be present from Bowl feeder. We might want to signal something in the light tower
	IF (StateTimer.Q) THEN
		Logging.fbEventMsg.SendEventMsg(MsgClass := TCEVENTCLASS_STATEINFO, EventID:= Logging.ID_CP_WaitCap, SourceID:= Logging.SrcCapPOU);
		StateTimer(IN:=FALSE);
		Status.CapStatusMsg:= 'No CAP from BOWL. Is Bowl ON?!!';
		NextState := eCapInsertStaState.eUnknown;
	END_IF    
	
	
eCapInsertStaState.eSendEscapementToPick:
   	GVL_IO.CP_YToolVacuumOFF:= TRUE;
    GVL_IO.CP_YToolVacuumON:= FALSE; 
   GVL_IO.CP_YEscapementToBowl := FALSE;
	GVL_IO.CP_YEscapementToPick := TRUE;	
	IF (NOT GVL_IO.CP_XEscapementAtBowl AND GVL_IO.CP_XEscapementAtPickUp) THEN
    		NextState := eCapInsertStaState.eEscapementAtPick;
	END_IF
	
	DwellTimer(IN:=TRUE, PT:= T#5S);
	IF (DwellTimer.Q) THEN
		NextState:= eCapInsertStaState.eInit;
		Logging.fbEventMsg.SendEventMsg(MsgClass := TCEVENTCLASS_STATEINFO, EventID:= Logging.ID_CP_CheckEscapeCylinders, SourceID:= Logging.SrcCapPOU);
		DwellTimer(IN:=FALSE);
		Status.CapStatusMsg:= 'Escapement NOT at Pick- CHECK JAMS, Clear and Hit Start!!';
		NextState := eCapInsertStaState.eUnknown;
	END_IF

eCapInsertStaState.eEscapementAtPick:    
	DwellTimer(IN:=TRUE, PT:= T#100MS);
	IF (DwellTimer.Q) THEN
	 NextState := eCapInsertStaState.eExtendWallCylinder;	
	 DwellTimer(IN:=FALSE);
	END_IF
     

eCapInsertStaState.eExtendWallCylinder:
    GVL_IO.CP_YEscapeWallCylinderExtend := TRUE;
	GVL_IO.CP_YEscapeWallCylinderRetract := FALSE;
	DwellTimer(IN:=TRUE, PT:= T#250MS);
	IF (DwellTimer.Q) THEN
		NextState := eCapInsertStaState.eRequestSMACCapPick;	 	
		DwellTimer(IN:=FALSE);
	END_IF	

eCapInsertStaState.eRequestSMACCapPick:
    GVL_IO.CP_YSMAC0 := FALSE;
	GVL_IO.CP_YSMAC1 := TRUE;
	GVL_IO.CP_YSMAC2 := FALSE;
	GVL_IO.CP_YSMAC3 := FALSE;
	DwellTimer(IN:=TRUE, PT:= T#50MS);	
	IF (DwellTimer.Q) THEN
		GVL_IO.CP_YSMAC3 := TRUE; // rising edge to trigger the selected SMAC routine every 5 seconds
		DwellTimer(IN:=FALSE);
		CapPickUpRetries := CapPickUpRetries + 1;
		NextState := eCapInsertStaState.eWaitForCapPickDone;
		StateTimer(IN:=FALSE);
	END_IF
	
eCapInsertStaState.eWaitForCapPickDone:
	DwellTimer(IN:=TRUE, PT:= T#150MS);
	IF (DwellTimer.Q) THEN
		IF (GVL_IO.CP_XSmac2 AND NOT GVL_IO.CP_XSmac1 AND GVL_IO.CP_XSmac0 ) THEN
			NextState := eCapInsertStaState.eTurnVacuumON;
			GVL_IO.CP_YSMAC3 := FALSE;
			DwellTimer(IN:=FALSE);
			CapPickUpRetries := 0;
		END_IF	
	END_IF   
	StateTimer(IN:=TRUE, PT:= T#4.5S); // SMAC timeouts in 5 seconds.
	IF (StateTimer.Q) THEN
		Logging.fbEventMsg.SendEventMsg(MsgClass := TCEVENTCLASS_STATEINFO, EventID:= Logging.ID_CP_MtrWaitCapPickCmpl, SourceID:= Logging.SrcCapPOU);
		StateTimer(IN:=FALSE);
		GVL_IO.CP_YSMAC3 := FALSE;		
		IF (CapPickupRetries < CONFIG.CAP_PICKUP_RETRIES ) THEN
			//NextState:=  eCapInsertStaState.eWallCylinderBackAndForth; // Operator check what the problem is and then hit the start button again; 
			  NextState := eCapInsertStaState.eRequestSMACCapPick; //Bonnie doesn't want the cyclinder wall to retract
              DwellTimer(IN:=FALSE);
 		ELSE
	    	NextState:= eCapInsertStaState.eUnknown ; // Operator check what the problem is and then hit the start button again;
			CapPickUpRetries := 0;
			Status.CapStatusMsg:= 'SMAC could not pick up CAP. Check CAP, then HIT START!!';
			NextState := eCapInsertStaState.eUnknown;
		END_IF		
	END_IF
	
eCapInsertStaState.eWallCylinderBackAndForth:
    GVL_IO.CP_YEscapeWallCylinderExtend := FALSE;
	GVL_IO.CP_YEscapeWallCylinderRetract := TRUE;
	DwellTimer(IN:=TRUE, PT:= T#250MS);
	IF (DwellTimer.Q) THEN		
		GVL_IO.CP_YEscapeWallCylinderExtend := TRUE;
		GVL_IO.CP_YEscapeWallCylinderRetract := FALSE;
		StateTimer(IN:= TRUE, PT := T#250MS);
		IF (StateTimer.Q) THEN        	
			NextState:= eCapInsertStaState.eRequestSMACCapPick;
			StateTimer(IN:=FALSE);
			DwellTimer(IN:=FALSE);
		END_IF
	END_IF
	
	
eCapInsertStaState.eTurnVacuumON:
	GVL_IO.CP_YToolVacuumON := TRUE;
	GVL_IO.CP_YToolVacuumOFF := FALSE;
	IF (GVL_IO.CP_XVacuumCapPicked) THEN
		NextState := eCapInsertStaState.eRetractWallCylinder; 
	END_IF
	DwellTimer(IN:=TRUE, PT:= T#150MS);
	IF (DwellTimer.Q) THEN
		//IF (GVL_IO.CP_XVacuumCapPicked) THEN
			NextState := eCapInsertStaState.eRetractWallCylinder; // do it anyways, because we aren't sure if the sensor is stable
			DwellTimer(IN:=FALSE);
	//	END_IF	
	END_IF   
	
eCapInsertStaState.eRetractWallCylinder:
	GVL_IO.CP_YEscapeWallCylinderExtend := FALSE;
	GVL_IO.CP_YEscapeWallCylinderRetract := TRUE;
	DwellTimer(IN:=TRUE, PT:= T#100MS);
	IF (DwellTimer.Q) THEN
		NextState := eCapInsertStaState.eRequestSMACHomeAfterPick;
		DwellTimer(IN:=FALSE); 	
	END_IF    
	

eCapInsertStaState.eRequestSMACHomeAfterPick:
    GVL_IO.CP_YSMAC0 := FALSE;
	GVL_IO.CP_YSMAC1 := FALSE;
	GVL_IO.CP_YSMAC2 := FALSE;
	GVL_IO.CP_YSMAC3 := FALSE;
	DwellTimer(IN:=TRUE, PT:= T#50MS);	
	IF (DwellTimer.Q) THEN
		GVL_IO.CP_YSMAC3 := TRUE; // rising edge to trigger the selected SMAC routine every 5 seconds
		DwellTimer(IN:=FALSE);
		NextState := eCapInsertStaState.eWaitForSMACHomeAfterPick;  	
	END_IF  

eCapInsertStaState.eWaitForSMACHomeAfterPick:	
	DwellTimer(IN:=TRUE, PT:= T#100MS);
	IF (DwellTimer.Q) THEN
		IF (GVL_IO.CP_XSmac2 AND GVL_IO.CP_XSmac1 AND GVL_IO.CP_XSmac0 ) THEN
			NextState := eCapInsertStaState.eSendEscapementToBowlNext;
			GVL_IO.CP_YSMAC3 := FALSE;
			DwellTimer(IN:=FALSE);
		END_IF	
	END_IF   
	StateTimer(IN:=TRUE, PT:= T#10S); // give a message out every 10 seconds
	IF (StateTimer.Q) THEN
		Logging.fbEventMsg.SendEventMsg(MsgClass := TCEVENTCLASS_STATEINFO, EventID:= Logging.ID_CP_MtrWaitReturnHomeCmpl, SourceID:= Logging.SrcCapPOU);
		StateTimer(IN:=FALSE);		
		NextState:= eCapInsertStaState.eUnknown; // Operator check what the problem is and then hit the start button again
		Status.CapStatusMsg:= 'SMAC Did not Home after PICK-- Check JAMS or is SMAC ON?!!';		
	END_IF
	

eCapInsertStaState.eSendEscapementToBowlNext:

	GVL_IO.CP_YEscapementToBowl := TRUE;
	GVL_IO.CP_YEscapementToPick := FALSE;
	IF (GVL_IO.CP_XEscapementAtBowl AND NOT GVL_IO.CP_XEscapementAtPickUp) THEN
    	NextState:= eCapInsertStaState.eEscapementAtBowlNext; 	
	END_IF
	
	StateTimer(IN:=TRUE, PT:= T#5S);
	IF (StateTimer.Q) THEN
		NextState:= eCapInsertStaState.eInit;
		Logging.fbEventMsg.SendEventMsg(MsgClass := TCEVENTCLASS_STATEINFO, EventID:= Logging.ID_CP_CheckEscapeCylinders, SourceID:= Logging.SrcCapPOU);
		StateTimer(IN:=FALSE);
		NextState:= eCapInsertStaState.eUnknown; // Operator check what the problem is and then hit the start button again
		Status.CapStatusMsg:= 'Escapement Did Not Get to Bowl Next.. Clear JAM and Hit START';
	END_IF

eCapInsertStaState.eEscapementatBowlNext:
   NextState := eCapInsertStaState.eWaitForVehicleTrigger;
	
eCapInsertStaState.eWaitForVehicleTrigger:
  
	IF (xTrigger) THEN //XTrigger is signaled when part arrives under the station
		
        NextState := eCapInsertStaState.ePalletHoldDownGoingDown;	
	    PartsData.Status[VUT].OverallStatus := ePartStatus.eReject; 		
		
		DwellTimer(IN:=FALSE);
	END_IF
	
	StateTimer(IN:=TRUE, PT:= T#10S); // give a message out every 10 seconds, hang out here indefinitely to wait for Parts to be present from Bowl feeder. We might want to signal something in the light tower
	IF (StateTimer.Q) THEN
		Logging.fbEventMsg.SendEventMsg(MsgClass := TCEVENTCLASS_STATEINFO, EventID:= Logging.ID_CP_WaitVehicle, SourceID:= Logging.SrcCapPOU);
		StateTimer(IN:=FALSE);
		Status.CapStatusMsg:= 'Waiting for CAP Part';
	END_IF


eCapInsertStaState.ePalletHoldDownGoingDown:
	GVL_IO.CP_YPalletHoldDownExtend := TRUE;
	GVL_IO.CP_YPalletHoldDownRetract := FALSE;
	IF (NOT GVL_IO.CP_XPalletHoldDownHome AND GVL_IO.CP_XPalletHoldDownExtended) THEN
		   NextState := eCapInsertStaState.ePalletHoldDownExtended;		   
	   END_IF
	
   DwellTimer(IN:=TRUE, PT:= T#1S); // give a message out every 10 seconds
	IF (DwellTimer.Q) THEN
		Logging.fbEventMsg.SendEventMsg(MsgClass := TCEVENTCLASS_STATEINFO, EventID:= Logging.ID_CP_CheckCylinders, SourceID:= Logging.SrcCapPOU);
		DwellTimer(IN:=FALSE);	
	END_IF
	StateTimer(IN:=TRUE, PT:= T#10S);  // if it is more than 10 seconds then we send the station into an unknown state and wait for operator to fix and hit start button again
	IF (StateTimer.Q) THEN
		Logging.fbEventMsg.SendEventMsg(MsgClass := TCEVENTCLASS_STATEINFO, EventID:= Logging.ID_CP_CheckCylinders, SourceID:= Logging.SrcCapPOU);
		StateTimer(IN:=FALSE);
		//NextState := eCapInsertStaState.ePalletHoldDownGoingUp; //move the vehicle out.. we need to notify the operator some kind of alarm here 
		NextState:= eCapInsertStaState.eUnknown; // Operator check what the problem is and then hit the start button again
		Status.CapStatusMsg:= 'Pallet Hold Down Not DOWN..check cyclinder/sensor then HIT START';
	END_IF  
   

eCapInsertStaState.ePalletHoldDownExtended:
   // NextState := eCapInsertStaState.eSendBarellCenterPinExtendRaise;
    NextState := eCapInsertStaState.eRequestSMACCapInstall;    // Skip the BarrelCenterPinExtend.
	CapInstallRetries := 0;

eCapInsertStaState.eSendBarellCenterPinExtendRaise:
	GVL_IO.CP_YBarellCenterPinExtend := TRUE;
	GVL_IO.CP_YBarellCenterPinRetract := FALSE;
	DwellTimer(IN:=FALSE);
	NextState := eCapInsertStaState.eCheckBarellCenterPinExtendedRaised;
	
	
eCapInsertStaState.eCheckBarellCenterPinExtendedRaised: // Note that these sensors are removed from the machine
    IF (NOT GVL_IO.CP_XBarellCenterPinRetracted AND GVL_IO.CP_XBarellCenterPinExtended) THEN
		DwellTimer(IN:= TRUE, PT := T#50MS);
		IF (DwellTimer.Q) THEN
			NextState := eCapInsertStaState.eRequestSMACCapInstall;
			DwellTimer(IN:=FALSE);			
		END_IF
	END_IF
	
	StateTimer(IN:=TRUE, PT:= T#10S);  // if it is more than 10 seconds then we send the station into an unknown state and wait for operator to fix and hit start button again
	IF (StateTimer.Q) THEN
		Logging.fbEventMsg.SendEventMsg(MsgClass := TCEVENTCLASS_STATEINFO, EventID:= Logging.ID_CP_CheckCylinders, SourceID:= Logging.SrcCapPOU);
		StateTimer(IN:=FALSE);
		NextState := eCapInsertStaState.ePalletHoldDownGoingUp; //move the vehicle out.. we need to notify the operator some kind of alarm here 
	END_IF  
	

eCapInsertStaState.eRequestSMACCapInstall:
    IF (LotsData.Lot.BarrelSize = eBarrelType.Size30cc) THEN
		GVL_IO.CP_YSMAC0 := TRUE; // shorter barrel
    ELSE
        GVL_IO.CP_YSMAC0 := FALSE; // longer barrel
	END_IF

	GVL_IO.CP_YSMAC1 := FALSE;
	GVL_IO.CP_YSMAC2 := TRUE;
	GVL_IO.CP_YSMAC3 := FALSE;
	DwellTimer(IN:=TRUE, PT:= T#50MS);	
	IF (DwellTimer.Q) THEN
		GVL_IO.CP_YSMAC3 := TRUE; // rising edge to trigger the selected SMAC routine every 5 seconds
		DwellTimer(IN:=FALSE);
		CapInstallRetries := CapInstallRetries +1;
		NextState := eCapInsertStaState.eWaitForSMACCapInstall;		
	END_IF

eCapInsertStaState.eWaitForSMACCapInstall:
	DwellTimer(IN:=TRUE, PT:= T#150MS);
	IF (DwellTimer.Q) THEN
		IF (GVL_IO.CP_XSmac2 AND GVL_IO.CP_XSmac1 AND NOT GVL_IO.CP_XSmac0 ) THEN
			UpdatePartData();
            NextState := eCapInsertStaState.eRequestSMACHome;
			GVL_IO.CP_YToolVacuumON := FALSE;
			GVL_IO.CP_YToolVacuumOFF := TRUE;
			GVL_IO.CP_YSMAC3 := FALSE;
			DwellTimer(IN:=FALSE);
		END_IF	
	END_IF   
	StateTimer(IN:=TRUE, PT:= T#7S); // give a message out every 10 seconds
	IF (StateTimer.Q) THEN
		Logging.fbEventMsg.SendEventMsg(MsgClass := TCEVENTCLASS_STATEINFO, EventID:= Logging.ID_CP_MtrWaitCapInsertCmpl, SourceID:= Logging.SrcCapPOU);
		StateTimer(IN:=FALSE);		
		GVL_IO.CP_YSMAC3 := FALSE;
		IF (CapInstallRetries < CONFIG.CAP_INSTALL_RETRIES) THEN
			NextState := eCapInsertStaState.eRequestSMACCapInstall;
		ELSE
			NextState := eCapInsertStaState.eRequestSMACHome;	 // keep Vacuum ON, we are going to reuse this cap on next part
            CapInstallRetries := 0;	
			//NextState:= eCapInsertStaState.eUnknown; // Operator check what the problem is and then hit the start button again
			 Status.CapStatusMsg:= 'SMAC Cap Install Timed OUT.. ';
		END_IF		
	END_IF

eCapInsertStaState.eRequestSMACHome:
    GVL_IO.CP_YSMAC0 := FALSE;
	GVL_IO.CP_YSMAC1 := FALSE;
	GVL_IO.CP_YSMAC2 := FALSE;
	GVL_IO.CP_YSMAC3 := FALSE;
	DwellTimer(IN:=TRUE, PT:= T#50MS);	
	IF (DwellTimer.Q) THEN
		GVL_IO.CP_YSMAC3 := TRUE; // rising edge to trigger the selected SMAC routine every 5 seconds
		DwellTimer(IN:=FALSE);
		NextState := eCapInsertStaState.eWaitForSMACHome;  	
	END_IF  

eCapInsertStaState.eWaitForSMACHome:	
	DwellTimer(IN:=TRUE, PT:= T#100MS);
	IF (DwellTimer.Q) THEN
		IF (GVL_IO.CP_XSmac2 AND GVL_IO.CP_XSmac1 AND GVL_IO.CP_XSmac0 ) THEN
			NextState := eCapInsertStaState.ePalletHoldDownGoingUp;
			GVL_IO.CP_YSMAC3 := FALSE;
			DwellTimer(IN:=FALSE);
		END_IF	
	END_IF   
	StateTimer(IN:=TRUE, PT:= T#15S); // give a message out every 10 seconds
	IF (StateTimer.Q) THEN
		Logging.fbEventMsg.SendEventMsg(MsgClass := TCEVENTCLASS_STATEINFO, EventID:= Logging.ID_CP_MtrWaitReturnHomeCmpl, SourceID:= Logging.SrcCapPOU);
		StateTimer(IN:=FALSE);		
		GVL_IO.CP_YSMAC3 := FALSE;
		//NextState:= eCapInsertStaState.ePalletHoldDownGoingUp; //Unknown; // Operator check what the problem is and then hit the start button again
		NextState:= eCapInsertStaState.eUnknown; // Operator check what the problem is and then hit the start button again
		Status.CapStatusMsg:= 'SMAC Could Not GO Home After CAP install.check for JAMS. Hit Start ';
	END_IF


eCapInsertStaState.ePalletHoldDownGoingUp:
   GVL_IO.CP_YPalletHoldDownExtend := FALSE;
   GVL_IO.CP_YPalletHoldDownRetract := TRUE;
   GVL_IO.CP_YBarellCenterPinExtend := FALSE;
   GVL_IO.CP_YBarellCenterPinRetract := TRUE;
   
   IF (GVL_IO.CP_XPalletHoldDownHome AND NOT GVL_IO.CP_XPalletHoldDownExtended (*AND  
       GVL_IO.CP_XBarellCenterPinRetracted AND NOT GVL_IO.CP_XBarellCenterPinExtended*)) THEN
	   NextState := eCapInsertStaState.ePalletHoldDownUp;
   END_IF
   
    DwellTimer(IN:=TRUE, PT:= T#1S); // give a message out every 10 seconds
	IF (DwellTimer.Q) THEN
		Logging.fbEventMsg.SendEventMsg(MsgClass := TCEVENTCLASS_STATEINFO, EventID:= Logging.ID_CP_CheckCylinders, SourceID:= Logging.SrcCapPOU);
		DwellTimer(IN:=FALSE);	
	END_IF
	StateTimer(IN:=TRUE, PT:= T#10S);  // if it is more than 10 seconds then we send the station into an unknown state and wait for operator to fix and hit start button again
	IF (StateTimer.Q) THEN
		Logging.fbEventMsg.SendEventMsg(MsgClass := TCEVENTCLASS_STATEINFO, EventID:= Logging.ID_CP_CheckCylinders, SourceID:= Logging.SrcCapPOU);
		StateTimer(IN:=FALSE);
		//NextState := eCapInsertStaState.eInit; //move the vehicle out.. we need to notify the operator some kind of alarm here 
		NextState:= eCapInsertStaState.eUnknown; // Operator check what the problem is and then hit the start button again
		Status.CapStatusMsg:= 'Pallet Hold Down Not Retracted. Check Cylinders then Press Start ';
	END_IF  

eCapInsertStaState.ePalletHoldDownUp:
   NextState := eCapInsertStaState.eDepart;

eCapInsertStaState.eDepart:
	Stations.fbRoutePlanner.M_NotifyVehStaCmpl(StationIndex:= MM_CONST.CAP_STA, VehicleID := VUT);
	xTrigger := FALSE; // Now that we have sent a vehicle out, we should not work on it anymore 
    IF (Stations.fbCycleControl.StopRequested) THEN		
		NextState := eCapInsertStaState.eStopActive;
	ELSE
		NextState := eCapInsertStaState.eHoming;
	END_IF

eCapInsertStaState.eStopActive:
IF (NOT Stations.fbCycleControl.StopRequested) THEN		
		NextState := eCapInsertStaState.eHoming;
END_IF	
    Status.CapStatusMsg:= 'Cap Stop Active, Press Start to Run';
	
eCapInsertStaState.eError:
END_CASE

IF (State <> NextState) THEN
	bFirst := TRUE;
	StateTimer(IN:=FALSE);
ELSE
	bFirst := FALSE;
END_IF

State := NextState;
AssignStationStatusForHMI();

METHOD PUBLIC AssignStationStatusForHMI : BOOL
VAR_INPUT
END_VAR
Status.StationsState[MM_CONST.CAP_STA_HMI_STATE] := State;
IF (NOT LotsData.Lot.CapInsertEnabled) THEN
	Status.StationStauts[MM_CONST.CAP_STA_HMI_STATE] := OverallStationStatus.eDisabled;
ELSE	
	CASE State OF
	eCapInsertStaState.eUnknown,eCapInsertStaState.eError: 
		Status.StationStauts[MM_CONST.CAP_STA_HMI_STATE] := OverallStationStatus.eError;
		
	eCapInsertStaState.eSMACMtrSendHome,eCapInsertStaState.eSMACMtrCheckHomed,eCapInsertStaState.eInit,eCapInsertStaState.eHoming,eCapInsertStaState.eReady,
	eCapInsertStaState.eSendEscapementToBowl,eCapInsertStaState.eSendEscapementToPick,eCapInsertStaState.eEscapementAtPick,
	eCapInsertStaState.eExtendWallCylinder, eCapInsertStaState.eRequestSMACCapPick,eCapInsertStaState.eWaitForCapPickDone,eCapInsertStaState.eWallCylinderBackAndForth,
	eCapInsertStaState.eTurnVacuumON,eCapInsertStaState.eRetractWallCylinder,eCapInsertStaState.eRequestSMACHomeAfterPick,eCapInsertStaState.eWaitForSMACHomeAfterPick,
	eCapInsertStaState.eSendEscapementToBowlNext,eCapInsertStaState.eEscapementatBowlNext:
	    Status.StationStauts[MM_CONST.CAP_STA_HMI_STATE] := OverallStationStatus.eHoming;
	
    eCapInsertStaState.eEscapementAtBowl:
	    Status.StationStauts[MM_CONST.CAP_STA_HMI_STATE] := OverallStationStatus.eWarning;
    
   eCapInsertStaState.eWaitForVehicleTrigger:
	    Status.StationStauts[MM_CONST.CAP_STA_HMI_STATE] := OverallStationStatus.eWaitingForParts;
	
    eCapInsertStaState.ePalletHoldDownGoingDown,eCapInsertStaState.ePalletHoldDownExtended,eCapInsertStaState.eSendBarellCenterPinExtendRaise,eCapInsertStaState.eCheckBarellCenterPinExtendedRaised,
	eCapInsertStaState.eRequestSMACCapInstall,eCapInsertStaState.eWaitForSMACCapInstall,eCapInsertStaState.eRequestSMACHome,eCapInsertStaState.eWaitForSMACHome,eCapInsertStaState.ePalletHoldDownGoingUp,
	eCapInsertStaState.ePalletHoldDownUp: 
	    Status.StationStauts[MM_CONST.CAP_STA_HMI_STATE] := OverallStationStatus.eRunning;
    
    eCapInsertStaState.eStopActive:
        Status.StationStauts[MM_CONST.CAP_STA_HMI_STATE] := OverallStationStatus.eCycleStop;	
   
    ELSE ;	
	END_CASE
END_IF
END_METHOD

METHOD PUBLIC ClearVehicleTrigger : BOOL
VAR_INPUT
END_VAR
xTrigger := FALSE;
END_METHOD

METHOD PUBLIC IsFaulted : BOOL
VAR_INPUT
END_VAR
IF (LotsData.Lot.CapInsertEnabled) THEN 
	IsFaulted := (State = eCapInsertStaState.eUnknown);
ELSE 
	IsFaulted := FALSE;
END_IF
END_METHOD

PROPERTY PUBLIC Ready : BOOL
GET
IF (LotsData.Lot.CapInsertEnabled) THEN
 Ready := (State = eCapInsertStaState.eWaitForVehicleTrigger);
ELSE
	Ready := TRUE;
 //Ready := (State = eCapInsertStaState.eDisabledReady);	//we removed the physical cap station on 10/17 
END_IF
END_GET
END_PROPERTY

METHOD PUBLIC ResetState : BOOL
VAR_INPUT
END_VAR
	State := eCapInsertStaState.eUnknown;
	NextState := eCapInsertStaState.eUnknown;
END_METHOD

PROPERTY PUBLIC Trigger : BOOL
SET
xTrigger := Trigger;
END_SET
END_PROPERTY

METHOD PUBLIC UpdatePartData : BOOL
VAR_INPUT
END_VAR
PartsData.Status[VUT].OverallStatus := ePartStatus.eCapInserted;
PartsData.Status[VUT].CapPass := TRUE;
PartsData.Status[VUT].CapInsertTime := SYSTEMTIME_TO_STRING(Logging.fbCurrTime.systemTime);
END_METHOD

PROPERTY PUBLIC VehicleUnderTest : BYTE
GET
VehicleUnderTest := VUT;
END_GET
SET
VUT := VehicleUnderTest;
END_SET
END_PROPERTY

END_FUNCTION_BLOCK

// ---- POUs/CheckBounds.TcPOU
// Implicitly generated code : DO NOT EDIT
FUNCTION CheckBounds : DINT
VAR_INPUT
	index, lower, upper: DINT;
END_VAR

// Implicitly generated code : Only an Implementation suggestion
{noflow}
IF  index < lower THEN
	CheckBounds := lower;
ELSIF  index > upper THEN
	CheckBounds := upper;
ELSE  
	CheckBounds := index;
END_IF
{flow}

END_FUNCTION
